TYPE ST_AddCommandIn :
STRUCT
	a		: REAL;
	b		: REAL;
END_STRUCT
END_TYPE

(* stored: Version 1.1.0.1, ProductVersion 3.1.4022.9
   DUT ST_AddCommandIn: Id {23bf6c56-d89b-48f9-8136-042134ff7447} *)
